FUNCTION_BLOCK FB_PIST
VAR_INPUT
	bInit: BOOL:=FALSE;
	open_time: TIME;
	close_time: TIME;
	open_timeout:TIME;
	close_timeout:TIME;
	eType: E_PIST_TYPE;
	bDefaultState: BOOL;
	bDepened_open1:BOOL:=TRUE;
	bDepened_open2:BOOL:=TRUE;
	bDepened_close1:BOOL:=TRUE;
	bDepened_close2:BOOL:=TRUE;
	sName:STRING;
END_VAR
VAR_OUTPUT
	pistStatus:E_PIST_STATUS:=E_PIST_STATUS.UNINIT ;
	bVALVE_OPEN: BOOL;
	bVALVE_CLOSE: BOOL;
	bError_Condition_open:BOOL;
	bError_Condition_close:BOOL;
	bERROR:BOOL:=FALSE;
END_VAR
VAR
	
	bCMD_OPEN: BOOL;
	bMANUAL: BOOL:=FALSE;
	bCMD_OPEN_SWR: BOOL;
	bCMD_CLOSE_SWR: BOOL;
	
	bSTARTUP: BOOL:=FALSE;
	bSEN_OPEN: BOOL;
	bSEN_CLOSE: BOOL;
	bStepDone: BOOL;
END_VAR

IF NOT bSTARTUP THEN
	bCMD_OPEN:=bDefaultState;
	bCMD_OPEN_SWR:=bDefaultState;
	bSTARTUP:=TRUE;
END_IF

IF NOT bMANUAL THEN
	bCMD_OPEN:=bCMD_OPEN_SWR;
END_IF

CASE pistStatus OF
	E_PIST_STATUS.UNINIT:
	IF bInit THEN
		pistStatus:=E_PIST_STATUS.INIT;
	END_IF
	
	E_PIST_STATUS.INIT:
	bInit:=FALSE;
	SFCReset:=TRUE;
	IF bCMD_OPEN THEN
		SFCReset:=FALSE;
		pistStatus:=E_PIST_STATUS.OPENING;
	ELSE
		SFCReset:=FALSE;
		pistStatus:=E_PIST_STATUS.CLOSING;
	END_IF
	
	E_PIST_STATUS.OPENING:
		open_pist();
		
	E_PIST_STATUS.CLOSING:
		close_pist();
	
	E_PIST_STATUS.OPENED:	
	IF NOT bCMD_OPEN THEN
		pistStatus:=E_PIST_STATUS.CLOSING;
	END_IF
	
	E_PIST_STATUS.CLOSED:	
	IF bCMD_OPEN THEN
		pistStatus:=E_PIST_STATUS.OPENING;
	END_IF
	
	E_PIST_STATUS.ERROR:
	IF bInit THEN
		pistStatus:=E_PIST_STATUS.INIT;
	END_IF

		
END_CASE

ACTION _aCHECK_active_1:
IF bDepened_open1 AND bDepened_open2 THEN
	bStepDone:=TRUE;
ELSE
	bError_Condition_open:=TRUE;
	pistStatus:=E_PIST_STATUS.ERROR;
	bERROR:=TRUE;
END_IF
END_ACTION

ACTION _aCHECK_active_1_1:
IF bDepened_close1 AND bDepened_close2 THEN
	bStepDone:=TRUE;
ELSE
	pistStatus:=E_PIST_STATUS.ERROR;
	bError_Condition_close:=FALSE;
	bERROR:=TRUE;
END_IF
END_ACTION

ACTION _aCHECK_entry:
bStepDone:=FALSE;
bERROR:=FALSE;
bError_Condition_open:=FALSE;
END_ACTION

ACTION _aCHECK_entry_1:
bStepDone:=FALSE;
bERROR:=FALSE;
bError_Condition_close:=FALSE;
END_ACTION

ACTION _aCLOSE_active:
IF eType=E_PIST_TYPE.NO_SENSORS OR eType=E_PIST_TYPE.ONLY_OPEN THEN
	IF CLOSE.t>close_time THEN
		bStepDone:=TRUE;
	END_IF
END_IF

	
IF eType=E_PIST_TYPE.BOTH OR eType=E_PIST_TYPE.ONLY_CLOSE THEN	
	IF bSEN_CLOSE THEN
		bStepDone:=TRUE;
	END_IF
	IF CLOSE.t>close_timeout THEN
		bERROR:=TRUE;
		bStepDone:=TRUE;
	END_IF
END_IF
END_ACTION

ACTION _aCLOSE_entry:
bStepDone:=FALSE;
bVALVE_CLOSE:=TRUE;
bVALVE_OPEN:=FALSE;
END_ACTION

ACTION _aCLOSE_exit:
IF NOT bERROR THEN
	pistStatus:=E_PIST_STATUS.CLOSED;
ELSE
	pistStatus:=E_PIST_STATUS.ERROR;
END_IF
END_ACTION

ACTION _aOPEN_active:
IF eType=E_PIST_TYPE.NO_SENSORS OR eType=E_PIST_TYPE.ONLY_CLOSE THEN
	IF OPEN.t>open_time THEN
		bStepDone:=TRUE;
	END_IF
END_IF

	
IF eType=E_PIST_TYPE.BOTH OR eType=E_PIST_TYPE.ONLY_OPEN THEN	
	IF bSEN_OPEN THEN
		bStepDone:=TRUE;
	END_IF
	IF OPEN.t>open_timeout THEN
		bERROR:=TRUE;
		bStepDone:=TRUE;
	END_IF
END_IF
END_ACTION

ACTION _aOPEN_entry:
bStepDone:=FALSE;
bVALVE_OPEN:=TRUE;
bVALVE_CLOSE:=FALSE;
END_ACTION

ACTION _aOPEN_exit:
IF NOT bERROR THEN
	pistStatus:=E_PIST_STATUS.OPENED;
ELSE
	pistStatus:=E_PIST_STATUS.ERROR;
END_IF
END_ACTION

ACTION A_CLOSE:
bCMD_OPEN_SWR:=FALSE;
END_ACTION

ACTION A_INIT:
bInit:=TRUE;
END_ACTION

ACTION A_OPEN:
bCMD_OPEN_SWR:=TRUE;
END_ACTION

ACTION close_pist:
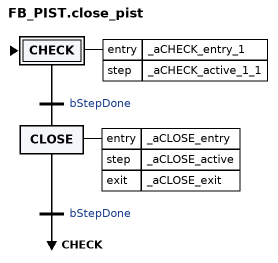
INITIAL_STEP CHECK:  // min time T#1s
    _aCHECK_entry_1(P1);  // entry action
    _aCHECK_active_1_1(N);  // step action
END_STEP
TRANSITION FROM CHECK TO CLOSE
    := bStepDone;
END_TRANSITION
STEP CLOSE:
    _aCLOSE_entry(P1);  // entry action
    _aCLOSE_active(N);  // step action
    _aCLOSE_exit(P0);  // exit action
END_STEP
TRANSITION FROM CLOSE TO CHECK
    := bStepDone;
END_TRANSITION
END_ACTION

ACTION open_pist:
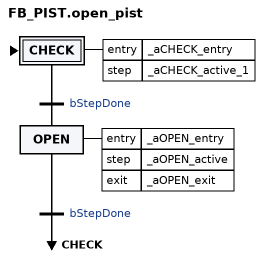
INITIAL_STEP CHECK:  // min time T#1s
    _aCHECK_entry(P1);  // entry action
    _aCHECK_active_1(N);  // step action
END_STEP
TRANSITION FROM CHECK TO OPEN
    := bStepDone;
END_TRANSITION
STEP OPEN:
    _aOPEN_entry(P1);  // entry action
    _aOPEN_active(N);  // step action
    _aOPEN_exit(P0);  // exit action
END_STEP
TRANSITION FROM OPEN TO CHECK
    := bStepDone;
END_TRANSITION
END_ACTION

END_FUNCTION_BLOCK

(* stored: Version 1.1.0.1, ProductVersion 3.1.4024.12
   POU FB_PIST: Id {d686fff2-be69-4be9-be07-961307b74eb8}, SpecialFunc None
   Action _aCHECK_active_1: Id {284b5af9-cde0-4865-9495-f3b272edbe9e}
   Action _aCHECK_active_1_1: Id {df789243-b467-4234-b6fc-624f388e7bd6}
   Action _aCHECK_entry: Id {fe1d960e-bcd7-4124-b49a-0ef3c820d872}
   Action _aCHECK_entry_1: Id {fc3e687d-f764-4ba5-bbe7-6af28bbd4082}
   Action _aCLOSE_active: Id {dec86915-94d9-4792-99d6-d46a5318759f}
   Action _aCLOSE_entry: Id {19d91e9b-25a3-4c14-bdc6-e600b00c5372}
   Action _aCLOSE_exit: Id {2ec6a691-8829-45d8-b599-498d07a33121}
   Action _aOPEN_active: Id {02819be6-7129-42a9-b3bb-2f875d412dc3}
   Action _aOPEN_entry: Id {82465bc6-834f-43a1-91a1-7e8224f8ef21}
   Action _aOPEN_exit: Id {867b2cf1-a166-458b-a99a-ad608a4e8e2d}
   Action A_CLOSE: Id {208f374d-f0e0-4104-ac27-2607f1b47699}
   Action A_INIT: Id {d8f097a9-85bd-44b3-9aef-23c87213367b}
   Action A_OPEN: Id {36193303-04ef-473d-b4cc-ee9b95d5e93c}
   Action close_pist: Id {a2391c5f-2c30-4fc8-a361-072a632167c7}
   Action open_pist: Id {963a9786-4727-40d2-b7a5-fddef60a1935} *)
